(* PLC project control_valve_52, Dassault Systèmes ControlBuild 2024x *)
(* stored: creationDateTime 2023-10-03T11:13:11-01:00 *)

(* This module simulates a five-way, two positions control valve used to drive a double-acting jack. *)
FUNCTION_BLOCK equipment_library.control_valve_52
  VAR_INPUT
    energy : BOOL := true;
    cmdSupply : BOOL := true;
  END_VAR
  VAR_INPUT
    valveWork : BOOL := false;
    valveRest : BOOL := false;
  END_VAR
  VAR_OUTPUT
    pipeWork : BOOL := false;
    pipeRest : BOOL := false;
  END_VAR
  VAR_OUTPUT
    workMode : BOOL := false;
    restMode : BOOL := false;
  END_VAR
  VAR
    slidePosition : DINT := 0;
  END_VAR
  VAR
    d_rest : BOOL := false;
    v_d_rest : BOOL := false;
    d_work : BOOL := false;
    v_d_work : BOOL := false;
  END_VAR


ACTION C_source_code:
/* ----------------------------------------------------------------	*/
/* Type : Model of Operative Behaviour					*/
/* Category :  Pre-actuators						*/
/* Author : Dassault Systemes						*/
/* Update date : June 2018							*/
/* ----------------------------------------------------------------	*/
/* This module simulates a five-way, two positions control valve	*/
/* used to drive a double-acting jack.					*/
/* ----------------------------------------------------------------	*/

/* ----------------------------------------------------------------	*/
/* Management of orders from Control Part					*/
/*	if there is no power supply for command the solenoid 		*/
/*     control valve doesn't understand the control order.		*/
/* Hypothesis : if the two control valves are excited at the 		*/
/* same time, only the first is taken into account.			*/
/* ----------------------------------------------------------------	*/
if (cmdSupply) {
	if (valveWork & ! valveRest) slidePosition = 1;
	if ( ! valveWork & valveRest) slidePosition = 0;
}

if (cmdSupply && valveWork) workMode = 1;
else workMode = 0;

if (cmdSupply && valveRest) restMode = 1;
else restMode = 0;

/* ----------------------------------------------------------------	*/
/* Calculation of the on-state of the energy in the pipes		*/
/*     if a fault is required on a pipe, the latter 			*/
/*		 takes a preset state.					*/
/*     if there is no energy in input, pipes are not 			*/
/*	   under pressure.							*/
/* ----------------------------------------------------------------	*/
if (d_work)
	pipeWork = v_d_work;
else
	pipeWork = (slidePosition==1) & energy;

if (d_rest)
	pipeRest = v_d_rest;
else
	pipeRest = (slidePosition==0) & energy;
END_ACTION
END_FUNCTION_BLOCK
